{attribute 'linkalways'} 
{attribute 'no_explicit_call' := 'This FB is a CLASS and must be accessed using methods or properties'}
{attribute 'enable_dynamic_creation'}
FUNCTION_BLOCK FINAL MUL_ULINT EXTENDS Node
VAR
	in1 : _ULINT(0);
	in2 : _ULINT(0);
	out : _ULINT(0);
END_VAR

METHOD PUBLIC Clone : I_Node
VAR
	pNode : POINTER TO MUL_ULINT;
END_VAR
pNode := __NEW(MUL_ULINT);
Clone := pNode^;
END_METHOD

METHOD FB_init : BOOL
VAR_INPUT
	bInitRetains : BOOL; // if TRUE, the retain variables are initialized (warm start / cold start)
	bInCopyCode : BOOL;  // if TRUE, the instance afterwards gets moved into the copy code (online change)
END_VAR
AddInput('in1',THIS^.in1);
AddInput('in2',THIS^.in2);
AddOutput('out', THIS^.out);
END_METHOD

METHOD PROTECTED OnExecute
VAR
END_VAR
out.Value := in1.Value * in2.Value;
END_METHOD

END_FUNCTION_BLOCK

(* stored: Version 1.1.0.1, ProductVersion 3.1.4024.15
   POU MUL_ULINT: Id {13a65333-df22-41b9-87f8-aa5c887f79a7}, SpecialFunc None
   Folder Constructor: Id {2a1ef629-4870-47f6-99ed-720c4c6ac79f}
   Method Clone: Id {c7c08b3d-6d05-4ee3-b28a-1cdceaf5c5f3}
   Method FB_init: Id {0f8ef700-186c-4059-8c6d-8601dafb77a6}
   Method OnExecute: Id {cff96d2f-09de-4196-a063-a06c29006648} *)
